Fanuc KAREL source: kc00038.KL

PROGRAM KC00038
%STACKSIZE=65535
%PRIORITY=65535
%NOLOCKGROUP
VAR
I : INTEGER
J : INTEGER
K : INTEGER
R : REAL
B : BOOLEAN
S : STRING[80]
T : STRING[80]
AI : ARRAY[8] OF INTEGER
JP : JOINTPOS9
AR : ARRAY[9] OF REAL
-- UNRESOLVED DECLARATIONS (source type spelling not recovered)
-- P : TYPE_0x001F (type_u16=0x001F)
-- Q : TYPE_0x001F (type_u16=0x001F)
-- AB : ARRAY[244] OF TYPE_0x0018 (type_u16=0x2018)
BEGIN
-- UNRESOLVED_PC line 18 opcodes [27 22 1C 22 22 76] marker_code=0
END KC00038
